// TIA Portal V16 export
// export: Created 2024-09-03T16:17:05.2198352Z, ExportSetting WithDefaults, DisplayName Totally Integrated Automation Portal, DisplayVersion V16, DisplayName TIA Portal Version Control Interface, DisplayVersion V16, DisplayName TIA Portal Openness, DisplayVersion V16, DisplayName STEP 7 Professional, DisplayVersion V16, DisplayName STEP 7 Safety, DisplayVersion V16, DisplayName WinCC Professional, DisplayVersion V16
DATA_BLOCK "DB00851_St_ConstAiScaleData"   // DB851
TITLE = Static DB [SYSTEM CONSTANTS] — Analog Input Scale Data and Ranges
{ S7_Optimized_Access := 'TRUE' }
AUTHOR : M_Gledhill
FAMILY : SysConstants
NAME : St_ConstAiScaleData
VERSION : 1.0
// PRACTICAL SERIES AUTOMATION LIBRARY (PAL)   —   COPYRIGHT 2020 – M. GLEDHILL (MIT LICENCE)
//                   ———— ◆ ————
// FULL ONLINE DOCUMENTATION IS AVAILABLE AT: https://practicalseries.com/2001-pal/index.html
// stored: AutoNumber false, DBAccessibleFromOPCUA true, IsOnlyStoredInLoadMemory false, IsRetainMemResEnabled false, IsWriteProtectedInAS false, MemoryReserve 100
   VAR
      _DB_Header { ExternalAccessible := 'False'; ExternalVisible := 'False'; ExternalWritable := 'False'} : Array[0..79] of Bool;   // Static DB [SYSTEM CONSTANTS] — Analog Input Scale Data and Ranges
      __________0000_0 { ExternalAccessible := 'False'; ExternalVisible := 'False'; ExternalWritable := 'False'} : Bool := false;
      __________0000_1 { ExternalAccessible := 'False'; ExternalVisible := 'False'; ExternalWritable := 'False'} : Bool := false;
      revInfo { ExternalWritable := 'False'} : "UT01000_St_SysRevision";
      __________0010_0 { ExternalAccessible := 'False'; ExternalVisible := 'False'; ExternalWritable := 'False'} : Bool := false;
      __________0010_1 { ExternalAccessible := 'False'; ExternalVisible := 'False'; ExternalWritable := 'False'} : Bool := false;   // ▀▀▀▀ ANALOG SCALE SIGNALS — TEST SIGNALS
      AI_SCALE_TST001 { ExternalWritable := 'False'; S7_SetPoint := 'True'} : "UT00851_Sy_ConstAiScaleData";   // Test range — 0 to 1000 l/s
      AI_SCALE_TST002 { ExternalWritable := 'False'; S7_SetPoint := 'True'} : "UT00851_Sy_ConstAiScaleData";   // Test range — -500 to +500 l/s
      AI_SCALE_TST003 { ExternalWritable := 'False'; S7_SetPoint := 'True'} : "UT00851_Sy_ConstAiScaleData";   // Test range — -1000 to 0 l/s
      AI_SCALE_TST004 { ExternalWritable := 'False'; S7_SetPoint := 'True'} : "UT00851_Sy_ConstAiScaleData";   // Test range — -270 to +1372 DegC
      AI_SCALE_TST005 { ExternalWritable := 'False'; S7_SetPoint := 'True'} : "UT00851_Sy_ConstAiScaleData";   // Test range — Erroneous configuration
      __________0020_0 { ExternalAccessible := 'False'; ExternalVisible := 'False'; ExternalWritable := 'False'} : Bool := false;
      __________0020_1 { ExternalAccessible := 'False'; ExternalVisible := 'False'; ExternalWritable := 'False'} : Bool := false;   // ▀▀▀▀ ANALOG SCALE SIGNALS — INSTRUMENTS
      AI_SCALE_TST006 { ExternalWritable := 'False'; S7_SetPoint := 'True'} : "UT00851_Sy_ConstAiScaleData";   // Test range — 0 to 1000 l/s
      AI_SCALE_FIC001 { ExternalWritable := 'False'; S7_SetPoint := 'True'} : "UT00851_Sy_ConstAiScaleData";   // Inlet flow meter (0-100 l/s)
      AI_SCALE_LIC001 { ExternalWritable := 'False'; S7_SetPoint := 'True'} : "UT00851_Sy_ConstAiScaleData";   // Inlet tank level (0-50 m3)
      AI_SCALE_PIC301 { ExternalWritable := 'False'; S7_SetPoint := 'True'} : "UT00851_Sy_ConstAiScaleData";   // Inlet filter differential pressure (0-2 BarG)
      AI_SCALE_PIC302 { ExternalWritable := 'False'; S7_SetPoint := 'True'} : "UT00851_Sy_ConstAiScaleData";   // Inlet filter differential pressure (0-2 BarG)
   END_VAR
BEGIN
   // _DB_Header[0] : ▄▄▄▄▄▄▄▄▄▄▄▄▄▄▄▄▄▄▄▄▄▄▄▄▄▄▄▄▄▄▄▄ ＣＯＮＳＴＡＮＴＳ ▄▄
   // _DB_Header[2] : TITLE: SYSTEM CONSTANTS — ANALOG INPUT SCALE DATA AND RANGES
   // _DB_Header[4] : ▀▀▀▀▀▀▀▀▀▀▀▀▀▀▀▀▀▀▀▀▀▀▀▀▀▀▀▀▀▀▀▀▀▀▀▀▀▀▀▀▀▀▀▀
   // _DB_Header[5] : TYPE: STATIC
   // _DB_Header[6] : ▄▄▄▄▄▄▄▄▄▄▄▄▄▄▄▄▄▄▄▄▄▄▄▄▄▄▄▄▄▄▄▄▄▄▄▄▄▄▄▄ ʷᴵᴰ⁻ᵈʰᵇ ▄
   // _DB_Header[8] : DB00851_St_ConstAiScaleData is a static data block that holds a full set of scaled ranges,
   // _DB_Header[9] : engineering units, device tag and descriptive data for all types of analog input scaled signals.
   // _DB_Header[11] : Each dataset is stored in a structure of user data type: UT00851_St_ConstAiScaleData.
   // _DB_Header[12] : This structure is configured to hold all the data required to name, scale and apply engineering
   // _DB_Header[13] : units to an analog input signal.
   // _DB_Header[15] : The scaled signal data is stored as constants and is used by all modules that have an interface
   // _DB_Header[16] : to an analog input card.
   // _DB_Header[18] : The purpose of the user data type and associated data block is to provide a consistent set of
   // _DB_Header[19] : scaled ranges and other data for each device or instrument that is available to the Controller
   // _DB_Header[20] : as an analog input.
   // _DB_Header[22] : The ranges correspond to the scaled values returned by the instrument or device, for example,
   // _DB_Header[23] : a flow meter may have a scaled range of -50 l/s to 200 l/s.
   // _DB_Header[25] : In addition, each dataset contains the instrument or device tag (e.g. FIC001), the engineering
   // _DB_Header[26] : units in use (e.g. l/s, kg/hour, °C, % &c.), over-range and under-range limits, a textual description
   // _DB_Header[27] : of the function of the instrument or device e.g. inlet flowmeter (0 l/s to 100 l/s) and additional
   // _DB_Header[28] : user specific information.
   // _DB_Header[30] : The PDF version of the SMDS for this module is available online here:
   // _DB_Header[31] : http://psop.uk/pal-smds-db00851-p
   // _DB_Header[33] : ━━━ ⬙⬙⬙⬙⬙⬙ ━━━
   // _DB_Header[35] : ▄▄▄▄▄▄▄▄▄▄▄▄▄▄▄▄▄▄▄▄▄▄▄▄▄▄▄▄▄▄▄▄▄▄▄▄▄▄▄▄▄▄▄▄
   // _DB_Header[36] : MODIFICATION HISTORY
   // _DB_Header[38] : This is a summary of the recent software modifications made to this block (most recent at top)
   // _DB_Header[40] : ―――――――――――――――――――――――――――――――――――――――――――
   // _DB_Header[41] : DATE REVISION MASTER BRANCH DEV
   // _DB_Header[42] : (nnn.amm) COMMIT TAG (Base ---> Merge) BRANCH Author
   // _DB_Header[43] : ———————————————————————————————————————————
   // _DB_Header[44] : 2022.05.15 001.000 D0018 D0017 D0018 None M. Gledhill
   // _DB_Header[45] : DB00851 — RELEASED FOR USE
   // _DB_Header[46] : Merge back to master branch
   // _DB_Header[48] : 2024.05.15 001.000 D0017A-000.104 D0017 N/A D0017A M. Gledhill
   // _DB_Header[49] : DB00851 — RELEASED FOR USE
   // _DB_Header[51] : 2024.05.03 000.801 D0017A-000.102 D0017 N/A D0017A M. Gledhill
   // _DB_Header[52] : DB00851 Block populated
   // _DB_Header[54] : 2024.04.09 000.101 D0017A-000.101 D0017 N/A D0017A M. Gledhill
   // _DB_Header[55] : DB00851 Block created
   // _DB_Header[56] : ———————————————————————————————————————————
   // _DB_Header[57] : Where: nnn = Major revision
   // _DB_Header[58] : a = Type (1-7 Development, 8 Proving, 9 Qualification, 0 Release)
   // _DB_Header[59] : mm = Minor revision (must be 00 if a = 0)
   // _DB_Header[60] : Block properties version number should be set to nn.a (only one decimal place)
   // _DB_Header[62] : ██████████████ █ █ █ █ END █ █ █ █ ██████████████
   revInfo.REV_BLOCK := 'DB00851';
   revInfo.REV_NUMBER := '001.000';
   revInfo.REV_DATE := '2024-05-15';
   revInfo.REV_AUTHOR := 'M. Gledhill';
   AI_SCALE_TST001.AI_TAG := 'TST001';
   AI_SCALE_TST001.SCALE_MIN := 0.0;
   AI_SCALE_TST001.SCALE_MAX := 1000.0;
   AI_SCALE_TST001.SCALE_UNITS := 'l/s';
   AI_SCALE_TST001.SCALE_DESC := 'Test Range (0 to 1000 l/s)';
   AI_SCALE_TST001.LIMIT_UNDER := -62.5;
   AI_SCALE_TST001.LIMIT_OVER := 1062.5;
   AI_SCALE_TST002.AI_TAG := 'TST002';
   AI_SCALE_TST002.SCALE_MIN := -500.0;
   AI_SCALE_TST002.SCALE_MAX := 500.0;
   AI_SCALE_TST002.SCALE_UNITS := 'l/s';
   AI_SCALE_TST002.SCALE_DESC := 'Test Range (-500 to 500 l/s)';
   AI_SCALE_TST002.LIMIT_UNDER := -562.5;
   AI_SCALE_TST002.LIMIT_OVER := 562.5;
   AI_SCALE_TST003.AI_TAG := 'TST003';
   AI_SCALE_TST003.SCALE_MIN := -1000.0;
   AI_SCALE_TST003.SCALE_MAX := 0.0;
   AI_SCALE_TST003.SCALE_UNITS := 'l/s';
   AI_SCALE_TST003.SCALE_DESC := 'Test Range (-1000 to 0 l/s)';
   AI_SCALE_TST003.LIMIT_UNDER := -1062.5;
   AI_SCALE_TST003.LIMIT_OVER := 62.5;
   AI_SCALE_TST004.AI_TAG := 'TST005';
   AI_SCALE_TST004.SCALE_MIN := -270.0;
   AI_SCALE_TST004.SCALE_MAX := 1372.0;
   AI_SCALE_TST004.SCALE_UNITS := 'DegC';
   AI_SCALE_TST004.SCALE_DESC := 'Test Range (-270 to +1372 DegC)';
   AI_SCALE_TST004.LIMIT_UNDER := -300.0;
   AI_SCALE_TST004.LIMIT_OVER := 1400.0;
   AI_SCALE_TST005.AI_TAG := 'TST005';
   AI_SCALE_TST005.___________0020_0 := false;
   AI_SCALE_TST005.___________0020_1 := false;
   AI_SCALE_TST005.SCALE_MIN := 0.0;
   AI_SCALE_TST005.SCALE_MAX := 1000.0;
   AI_SCALE_TST005.SCALE_UNITS := 'l/s';
   AI_SCALE_TST005.SCALE_DESC := 'Test Range (0 to 1000 l/s)';
   AI_SCALE_TST005.___________0030_0 := false;
   AI_SCALE_TST005.___________0030_1 := false;
   AI_SCALE_TST005.LIMIT_UNDER := 100.0;
   AI_SCALE_TST005.LIMIT_OVER := 900.0;
   AI_SCALE_TST006.AI_TAG := 'TST005';
   AI_SCALE_TST006.SCALE_MIN := 0.0;
   AI_SCALE_TST006.SCALE_MAX := 1000.0;
   AI_SCALE_TST006.SCALE_UNITS := 'l/s';
   AI_SCALE_TST006.SCALE_DESC := 'Test Range (0 to 1000 l/s)';
   AI_SCALE_TST006.LIMIT_UNDER := 100.0;
   AI_SCALE_TST006.LIMIT_OVER := 900.0;
   AI_SCALE_FIC001.AI_TAG := 'FIC001';
   AI_SCALE_FIC001.SCALE_MIN := 0.0;
   AI_SCALE_FIC001.SCALE_MAX := 100.0;
   AI_SCALE_FIC001.SCALE_UNITS := 'l/s';
   AI_SCALE_FIC001.SCALE_DESC := 'Inlet flow meter (0-100 l/s)';
   AI_SCALE_FIC001.LIMIT_UNDER := -5.0;
   AI_SCALE_FIC001.LIMIT_OVER := 105.0;
   AI_SCALE_FIC001.USER_INFO_1 := 'Instrument manufacturer: Siemens';
   AI_SCALE_FIC001.USER_INFO_2 := 'Instrument type: Sitrans FM MAG 5000 (mass flow)';
   AI_SCALE_FIC001.USER_INFO_3 := 'Instrument part no.: 7ME5920-1AA10-1AA0';
   AI_SCALE_FIC001.USER_INFO_4 := 'Instrument serial no.: 3443201102';
   AI_SCALE_LIC001.AI_TAG := 'LIC001';
   AI_SCALE_LIC001.SCALE_MIN := 0.0;
   AI_SCALE_LIC001.SCALE_MAX := 50.0;
   AI_SCALE_LIC001.SCALE_UNITS := 'm3';
   AI_SCALE_LIC001.SCALE_DESC := 'Inlet tank level (0-50 m3)';
   AI_SCALE_LIC001.LIMIT_UNDER := -2.5;
   AI_SCALE_LIC001.LIMIT_OVER := 52.5;
   AI_SCALE_LIC001.USER_INFO_1 := 'Instrument manufacturer: Siemens';
   AI_SCALE_LIC001.USER_INFO_2 := 'Instrument type: Sitrans LU240 (level)';
   AI_SCALE_LIC001.USER_INFO_3 := 'Instrument part no.: 7ML5110-1DD07-4AF0';
   AI_SCALE_LIC001.USER_INFO_4 := 'Instrument serial no.: 4514461005';
   AI_SCALE_PIC301.AI_TAG := 'PIC301';
   AI_SCALE_PIC301.SCALE_MIN := 0.0;
   AI_SCALE_PIC301.SCALE_MAX := 2.0;
   AI_SCALE_PIC301.SCALE_UNITS := 'BarG';
   AI_SCALE_PIC301.SCALE_DESC := 'Inlet filter differential pressure (0-2 BarG)';
   AI_SCALE_PIC301.LIMIT_UNDER := -0.1;
   AI_SCALE_PIC301.LIMIT_OVER := 2.1;
   AI_SCALE_PIC301.USER_INFO_1 := 'Instrument manufacturer: Siemens';
   AI_SCALE_PIC301.USER_INFO_2 := 'Instrument type: Sitrans P420 (pressure)';
   AI_SCALE_PIC301.USER_INFO_3 := 'Instrument part no.: 7MF0440-1ML02-5BF0';
   AI_SCALE_PIC301.USER_INFO_4 := 'Instrument serial no.: 7875344001';
   AI_SCALE_PIC302.AI_TAG := 'PIC301';
   AI_SCALE_PIC302.SCALE_MIN := 0.0;
   AI_SCALE_PIC302.SCALE_MAX := 2.0;
   AI_SCALE_PIC302.SCALE_UNITS := 'BarG';
   AI_SCALE_PIC302.SCALE_DESC := 'Inlet filter differential pressure (0-2 BarG)';
   AI_SCALE_PIC302.LIMIT_UNDER := -0.1;
   AI_SCALE_PIC302.LIMIT_OVER := 2.1;
   AI_SCALE_PIC302.USER_INFO_1 := 'Instrument manufacturer: Siemens';
   AI_SCALE_PIC302.USER_INFO_2 := 'Instrument type: Sitrans P420 (pressure)';
   AI_SCALE_PIC302.USER_INFO_3 := 'Instrument part no.: 7MF0440-1ML02-5BF0';
   AI_SCALE_PIC302.USER_INFO_4 := 'Instrument serial no.: 7875344008';
END_DATA_BLOCK
